TYPE ST_System_HS_Zustand :
STRUCT
	Betrieb_Anford				: BOOL;
	Betrieb_Soll				: BOOL;
	Betrieb						: BOOL;
	Betrieb_Kennlinie			: BOOL;

	Regelung_Modus				: SINT;
	Regelung_Sollw				: REAL;

	Freigabe					: BOOL;
	Freigabe_Deakt				: BOOL;
	Freigabe_Code				: WORD;

	Modus_eingeschaltet			: BOOL;
	Modus_ausgeschaltet			: BOOL;

	Stoerung					: BOOL;
	Stoerung_Code				: WORD;

	Warnung						: BOOL;
	Warnung_Code				: WORD;

	Status						: SINT;
	Temp_Regelungswert			: REAL;

	Quittierung					: BOOL;
END_STRUCT
END_TYPE

(* stored: Version 1.1.0.1, ProductVersion 3.1.4024.9
   DUT ST_System_HS_Zustand: Id {b6adac87-d375-4752-a00b-a0f2bdaac432} *)
